// Implicitly generated code : DO NOT EDIT
FUNCTION CheckDivDInt : DINT
VAR_INPUT
	divisor:DINT;
END_VAR

// Implicitly generated code : Only an Implementation suggestion
{noflow}
IF divisor = 0 THEN
	G_Diag.uiCheckDivDint:=G_Diag.uiCheckDivDint+1;
	CheckDivDInt:=1;
ELSE
	CheckDivDInt:=divisor;
END_IF;
{flow}

END_FUNCTION

(* stored: Version 1.1.0.1, ProductVersion 3.1.4024.4
   POU CheckDivDInt: Id {a66ac02f-7d5c-4ee2-8a8a-2f984461974e}, SpecialFunc CheckDivInt32 *)
